(* IEC 61131-3 sources: plc-workspace/projects/FB_MainSequence/03_checks/openplc, 2 files *)

(* ---- FB_MainSequence_OpenPLC.st ---- *)
(* Generated by validation/scripts/sync-semantics.py; edit 02_src/st. *)
FUNCTION FC_MainSequence_BusyPhase : BOOL
VAR_INPUT
    iPhase : INT := 0;
END_VAR

FC_MainSequence_BusyPhase := (iPhase = 1) OR (iPhase = 2) OR (iPhase = 3);

END_FUNCTION

FUNCTION FC_MainSequence_InvalidPhase : BOOL
VAR_INPUT
    iPhase : INT := 0;
END_VAR

FC_MainSequence_InvalidPhase := (iPhase < 0) OR ((iPhase > 3) AND (iPhase <> 900));

END_FUNCTION

FUNCTION FC_MainSequence_StepDone : BOOL
VAR_INPUT
    iPhase : INT := 0;
    xTransportDone : BOOL := FALSE;
    xFlipDone : BOOL := FALSE;
    xOutputDone : BOOL := FALSE;
END_VAR

CASE iPhase OF
    1:
        FC_MainSequence_StepDone := xTransportDone;
    2:
        FC_MainSequence_StepDone := xFlipDone;
    3:
        FC_MainSequence_StepDone := xOutputDone;
    ELSE
        FC_MainSequence_StepDone := FALSE;
END_CASE;

END_FUNCTION

FUNCTION FC_MainSequence_SuccessPhase : INT
VAR_INPUT
    iPhase : INT := 0;
END_VAR

CASE iPhase OF
    1:
        FC_MainSequence_SuccessPhase := 2;
    2:
        FC_MainSequence_SuccessPhase := 3;
    3:
        FC_MainSequence_SuccessPhase := 1;
    ELSE
        FC_MainSequence_SuccessPhase := iPhase;
END_CASE;

END_FUNCTION

FUNCTION FC_MainSequence_TimeoutReached : BOOL
VAR_INPUT
    xBusyPhase : BOOL := FALSE;
    xStepDone : BOOL := FALSE;
    uiStepTimerStat : UINT := 0;
    uiStepTimeoutScans : UINT := 0;
END_VAR

FC_MainSequence_TimeoutReached :=
    xBusyPhase AND
    (NOT xStepDone) AND
    (uiStepTimeoutScans > 0) AND
    ((uiStepTimerStat + 1) >= uiStepTimeoutScans);

END_FUNCTION

FUNCTION FC_MainSequence_NextPhase : INT
VAR_INPUT
    xClearReq : BOOL := FALSE;
    xAbortReq : BOOL := FALSE;
    xFaultLatched : BOOL := FALSE;
    iPhaseStat : INT := 0;
    xInvalidPhase : BOOL := FALSE;
    xStepDone : BOOL := FALSE;
    xTimeoutReached : BOOL := FALSE;
    iSuccessPhase : INT := 0;
    xStartReady : BOOL := FALSE;
END_VAR

IF xClearReq THEN
    FC_MainSequence_NextPhase := 0;
ELSIF xFaultLatched OR xInvalidPhase THEN
    FC_MainSequence_NextPhase := 900;
ELSIF xAbortReq THEN
    FC_MainSequence_NextPhase := 0;
ELSIF iPhaseStat = 0 THEN
    IF xStartReady THEN
        FC_MainSequence_NextPhase := 1;
    ELSE
        FC_MainSequence_NextPhase := 0;
    END_IF;
ELSIF iPhaseStat = 900 THEN
    FC_MainSequence_NextPhase := 900;
ELSIF xInvalidPhase THEN
    FC_MainSequence_NextPhase := 900;
ELSIF xStepDone THEN
    FC_MainSequence_NextPhase := iSuccessPhase;
ELSIF xTimeoutReached THEN
    FC_MainSequence_NextPhase := 900;
ELSE
    FC_MainSequence_NextPhase := iPhaseStat;
END_IF;

END_FUNCTION

FUNCTION FC_MainSequence_NextTimer : UINT
VAR_INPUT
    xResetReq : BOOL := FALSE;
    iPhaseStat : INT := 0;
    xInvalidPhase : BOOL := FALSE;
    xStepDone : BOOL := FALSE;
    xTimeoutReached : BOOL := FALSE;
    xBusyPhase : BOOL := FALSE;
    uiStepTimerStat : UINT := 0;
    uiStepTimeoutScans : UINT := 0;
END_VAR

IF xResetReq OR (iPhaseStat = 0) OR (iPhaseStat = 900) OR xInvalidPhase OR xStepDone OR xTimeoutReached THEN
    FC_MainSequence_NextTimer := 0;
ELSIF xBusyPhase AND (uiStepTimeoutScans > 0) THEN
    FC_MainSequence_NextTimer := uiStepTimerStat + 1;
ELSE
    FC_MainSequence_NextTimer := 0;
END_IF;

END_FUNCTION

FUNCTION FC_MainSequence_NextTimeoutFault : BOOL
VAR_INPUT
    xClearReq : BOOL := FALSE;
    xAbortReq : BOOL := FALSE;
    xTimeoutReached : BOOL := FALSE;
    xTimeoutFaultStat : BOOL := FALSE;
END_VAR

IF xClearReq THEN
    FC_MainSequence_NextTimeoutFault := FALSE;
ELSIF xAbortReq THEN
    FC_MainSequence_NextTimeoutFault := xTimeoutFaultStat;
ELSE
    FC_MainSequence_NextTimeoutFault := xTimeoutFaultStat OR xTimeoutReached;
END_IF;

END_FUNCTION

FUNCTION_BLOCK FB_MainSequence
VAR_INPUT
    xEnable : BOOL := FALSE;
    xEvtStart : BOOL := FALSE;
    xEStop : BOOL := FALSE;
    xStop : BOOL := FALSE;
    xReset : BOOL := FALSE;
    xInitDone : BOOL := FALSE;
    xTransportDone : BOOL := FALSE;
    xFlipDone : BOOL := FALSE;
    xOutputDone : BOOL := FALSE;
    uiStepTimeoutScans : UINT := 8;
END_VAR

VAR_OUTPUT
    iPhase : INT := 0;
    xBeltForward : BOOL := FALSE;
    xBeltReverse : BOOL := FALSE;
    xStartLamp : BOOL := FALSE;
    xResetLamp : BOOL := FALSE;
    xQ1 : BOOL := FALSE;
    xQ2 : BOOL := FALSE;
    xDone : BOOL := FALSE;
    xError : BOOL := FALSE;
    xTimeoutFault : BOOL := FALSE;
    xValid : BOOL := FALSE;
    xBusy : BOOL := FALSE;
    xCommandBusy : BOOL := FALSE;
    xCommandAborted : BOOL := FALSE;
    xTimeoutDiagnostic : BOOL := FALSE;
END_VAR

VAR
    iPhaseStat : INT := 0;
    uiStepTimerStat : UINT := 0;
    xTimeoutFaultStat : BOOL := FALSE;
    xTimeoutDiagnosticStat : BOOL := FALSE;
    xAbortedStat : BOOL := FALSE;
    xEnablePrev : BOOL := FALSE;
    xStartPrev : BOOL := FALSE;
    xResetPrev : BOOL := FALSE;
END_VAR

VAR_TEMP
    iPhasePrev : INT;
    uiStepTimerPrev : UINT;
    xTimeoutFaultPrev : BOOL;
    xDiagnosticPrev : BOOL;
    xAbortedPrev : BOOL;
    xEnableRise : BOOL;
    xStartRise : BOOL;
    xResetRise : BOOL;
    xStopReq : BOOL;
    xResetAccepted : BOOL;
    xClearReq : BOOL;
    xAbortReq : BOOL;
    xInvalidPhase : BOOL;
    xBusyPhase : BOOL;
    xFaultLatched : BOOL;
    xStepDone : BOOL;
    xTimeoutReached : BOOL;
    iPhaseNext : INT;
    uiStepTimerNext : UINT;
    xTimeoutFaultNext : BOOL;
    xDiagnosticNext : BOOL;
    xAbortedNext : BOOL;
    xStartAccepted : BOOL;
    xErrorCore : BOOL;
    xExecAllowed : BOOL;
END_VAR

(* Snapshot persistent internals only; outputs are never used as state. *)
iPhasePrev := iPhaseStat;
uiStepTimerPrev := uiStepTimerStat;
xTimeoutFaultPrev := xTimeoutFaultStat;
xDiagnosticPrev := xTimeoutDiagnosticStat;
xAbortedPrev := xAbortedStat;
xEnableRise := xEnable AND NOT xEnablePrev;
xStartRise := xEvtStart AND NOT xStartPrev;
xResetRise := xReset AND NOT xResetPrev;

(* xEStop is external safety-inhibit feedback, not an F safety function.
   Reset reinitializes a healthy command. Block errors need enable=FALSE. *)
xStopReq := xEStop OR xStop;
xInvalidPhase := FC_MainSequence_InvalidPhase(iPhase := iPhasePrev);
xBusyPhase := FC_MainSequence_BusyPhase(iPhase := iPhasePrev);
xFaultLatched := (iPhasePrev = 900) OR xTimeoutFaultPrev;
xResetAccepted := xEnable AND xResetRise AND NOT xStopReq AND NOT xFaultLatched AND NOT xInvalidPhase;
xClearReq := (NOT xEnable) OR xResetAccepted;
xAbortReq := xStopReq OR xReset;
xStepDone := FC_MainSequence_StepDone(
    iPhase := iPhasePrev,
    xTransportDone := xTransportDone,
    xFlipDone := xFlipDone,
    xOutputDone := xOutputDone
);
xTimeoutReached := FC_MainSequence_TimeoutReached(
    xBusyPhase := xBusyPhase,
    xStepDone := xStepDone,
    uiStepTimerStat := uiStepTimerPrev,
    uiStepTimeoutScans := uiStepTimeoutScans
);

iPhaseNext := FC_MainSequence_NextPhase(
    xClearReq := xClearReq,
    xAbortReq := xAbortReq,
    xFaultLatched := xFaultLatched,
    iPhaseStat := iPhasePrev,
    xInvalidPhase := xInvalidPhase,
    xStepDone := xStepDone,
    xTimeoutReached := xTimeoutReached,
    iSuccessPhase := FC_MainSequence_SuccessPhase(iPhase := iPhasePrev),
    xStartReady := xEnable AND xInitDone AND xStartRise
);
uiStepTimerNext := FC_MainSequence_NextTimer(
    xResetReq := xClearReq OR xAbortReq,
    iPhaseStat := iPhasePrev,
    xInvalidPhase := xInvalidPhase,
    xStepDone := xStepDone,
    xTimeoutReached := xTimeoutReached,
    xBusyPhase := xBusyPhase,
    uiStepTimerStat := uiStepTimerPrev,
    uiStepTimeoutScans := uiStepTimeoutScans
);
xTimeoutFaultNext := FC_MainSequence_NextTimeoutFault(
    xClearReq := xClearReq,
    xAbortReq := xAbortReq,
    xTimeoutReached := xTimeoutReached,
    xTimeoutFaultStat := xTimeoutFaultPrev
);
xStartAccepted := (iPhasePrev = 0) AND (iPhaseNext = 1);

(* Current errors and diagnostic history have separate lifetimes. *)
IF xEnableRise THEN
    xDiagnosticNext := xTimeoutFaultNext;
ELSE
    xDiagnosticNext := xDiagnosticPrev OR xTimeoutFaultNext;
END_IF;
IF xBusyPhase AND (xClearReq OR xAbortReq) THEN
    xAbortedNext := TRUE;
ELSIF (NOT xEnable) OR xResetAccepted OR xStartAccepted THEN
    xAbortedNext := FALSE;
ELSE
    xAbortedNext := xAbortedPrev;
END_IF;
xErrorCore := FC_MainSequence_InvalidPhase(iPhase := iPhaseNext) OR (iPhaseNext = 900);
xExecAllowed := xEnable AND NOT xAbortReq AND NOT xErrorCore;

(* Commit once. Consume input edges on every call, even while inhibited. *)
iPhaseStat := iPhaseNext;
uiStepTimerStat := uiStepTimerNext;
xTimeoutFaultStat := xTimeoutFaultNext;
xTimeoutDiagnosticStat := xDiagnosticNext;
xAbortedStat := xAbortedNext;
xEnablePrev := xEnable;
xStartPrev := xEvtStart;
xResetPrev := xReset;

(* DA008: each output is assigned once and no output is read. *)
iPhase := iPhaseNext;
xError := xErrorCore;
xTimeoutFault := xTimeoutFaultNext;
xBeltForward := xExecAllowed AND ((iPhaseNext = 1) OR (iPhaseNext = 3));
xBeltReverse := FALSE;
xStartLamp := xExecAllowed AND ((iPhaseNext = 2) OR (iPhaseNext = 3));
xResetLamp := xExecAllowed AND (iPhaseNext = 0);
xQ1 := xExecAllowed AND (iPhaseNext = 2);
xQ2 := xExecAllowed AND (iPhaseNext = 3);
xDone := xExecAllowed AND (iPhasePrev = 3) AND xOutputDone AND (iPhaseNext = 1);
xValid := xEnable AND NOT xErrorCore;
xBusy := xEnable AND NOT xErrorCore;
xCommandBusy := xExecAllowed AND FC_MainSequence_BusyPhase(iPhase := iPhaseNext);
xCommandAborted := xAbortedNext;
xTimeoutDiagnostic := xDiagnosticNext;

END_FUNCTION_BLOCK

(* OpenPLC-only test driver. Core definitions are generated from 02_src/st. *)
PROGRAM PLC_PRG
VAR
    fbMain : FB_MainSequence;
    xEnableSim : BOOL := TRUE;
    xEvtStartSim : BOOL := FALSE;
    xEStopSim : BOOL := FALSE;
    xResetSim : BOOL := FALSE;
    xInitDoneSim : BOOL := TRUE;
    xTransportDoneSim : BOOL := FALSE;
    xFlipDoneSim : BOOL := FALSE;
    xOutputDoneSim : BOOL := FALSE;
    uiStepTimeoutScansSim : UINT := 8;

    iObservedPhase : INT := 0;
    xObservedDone : BOOL := FALSE;
    xObservedError : BOOL := FALSE;
    xObservedTimeoutFault : BOOL := FALSE;

    iLastObservedPhase : INT := -1;
    iPhaseDwell : INT := 0;
    iCycleCountInternal : INT := 0;
    iResetCountInternal : INT := 0;
    iScanCountInternal : INT := 0;
    iScenarioCaseInternal : INT := 0;
    iNextScenarioAfterReset : INT := -1;
    iErrorPhaseLatched : INT := 0;

    xDoneLast : BOOL := FALSE;
    xResetPending : BOOL := FALSE;
    xStartPulsePending : BOOL := FALSE;
    xFaultScenarioStarted : BOOL := FALSE;
    xFaultPulseIssued : BOOL := FALSE;
    xRepeatScenarioStarted : BOOL := FALSE;
    iRepeatPulseCount : INT := 0;
    iRepeatBaselineCycle : INT := -1;
    xTimeoutScenarioStarted : BOOL := FALSE;
    xDisablePending : BOOL := FALSE;
END_VAR

VAR
    iPhaseMon AT %MW0 : INT;
    iCycleCountMon AT %MW1 : INT;
    iResetCountMon AT %MW2 : INT;
    iScanCountMon AT %MW3 : INT;
    iScenarioCaseMon AT %MW4 : INT;
    iErrorPhaseMon AT %MW5 : INT;

    xSawPhase0Mon AT %QX0.0 : BOOL;
    xSawPhase1Mon AT %QX0.1 : BOOL;
    xSawPhase2Mon AT %QX0.2 : BOOL;
    xSawPhase3Mon AT %QX0.3 : BOOL;
    xSawDoneMon AT %QX0.4 : BOOL;
    xSawResetReturnMon AT %QX0.5 : BOOL;
    xBehaviorPassMon AT %QX0.6 : BOOL;
    xBehaviorFailMon AT %QX0.7 : BOOL;

    xFaultInterruptPassMon AT %QX1.0 : BOOL;
    xRepeatStartBlockedPassMon AT %QX1.1 : BOOL;
    xTimeoutFailPassMon AT %QX1.2 : BOOL;
    xStartEventRequiredPassMon AT %QX1.3 : BOOL;
    xTimeoutErrorPassMon AT %QX1.4 : BOOL;
END_VAR

iScanCountInternal := iScanCountInternal + 1;
xEvtStartSim := FALSE;
xEStopSim := FALSE;
xResetSim := FALSE;
xTransportDoneSim := FALSE;
xFlipDoneSim := FALSE;
xOutputDoneSim := FALSE;
xEnableSim := TRUE;
xInitDoneSim := TRUE;

IF xDisablePending THEN
    xEnableSim := FALSE;
    xDisablePending := FALSE;
END_IF;

IF xResetPending THEN
    xResetSim := TRUE;
    xResetPending := FALSE;
    iResetCountInternal := iResetCountInternal + 1;
END_IF;

IF xStartPulsePending THEN
    xEvtStartSim := TRUE;
    xStartPulsePending := FALSE;
END_IF;

IF iScenarioCaseInternal = 99 THEN
    xEnableSim := FALSE;
    xInitDoneSim := FALSE;
END_IF;

CASE iScenarioCaseInternal OF
    0:
        IF (iObservedPhase <> 0) AND (NOT xStartEventRequiredPassMon) AND (iCycleCountInternal = 0) THEN
            xBehaviorFailMon := TRUE;
        END_IF;
        IF (iObservedPhase = 0) AND (iPhaseDwell >= 2) AND (NOT xStartEventRequiredPassMon) THEN
            xStartEventRequiredPassMon := TRUE;
            xStartPulsePending := TRUE;
            iScenarioCaseInternal := 1;
        END_IF;

    1:
        CASE iLastObservedPhase OF
            1:
                IF iPhaseDwell >= 2 THEN
                    xTransportDoneSim := TRUE;
                END_IF;
            2:
                IF iPhaseDwell >= 2 THEN
                    xFlipDoneSim := TRUE;
                END_IF;
            3:
                IF iPhaseDwell >= 2 THEN
                    xOutputDoneSim := TRUE;
                END_IF;
        END_CASE;

    2:
        IF (NOT xFaultScenarioStarted) AND (iObservedPhase = 0) AND (iPhaseDwell >= 1) THEN
            xStartPulsePending := TRUE;
            xFaultScenarioStarted := TRUE;
        END_IF;
        IF xFaultScenarioStarted AND (iObservedPhase = 1) AND (iPhaseDwell >= 2) AND (NOT xFaultPulseIssued) THEN
            xEStopSim := TRUE;
            xFaultPulseIssued := TRUE;
        END_IF;

    3:
        IF (NOT xRepeatScenarioStarted) AND (iObservedPhase = 0) AND (iPhaseDwell >= 1) THEN
            xStartPulsePending := TRUE;
            xRepeatScenarioStarted := TRUE;
        END_IF;

        CASE iLastObservedPhase OF
            1:
                IF iPhaseDwell >= 2 THEN
                    xTransportDoneSim := TRUE;
                END_IF;
            2:
                IF iRepeatBaselineCycle < 0 THEN
                    iRepeatBaselineCycle := iCycleCountInternal;
                END_IF;
                IF (iRepeatPulseCount < 3) AND (iPhaseDwell >= (iRepeatPulseCount + 1)) THEN
                    xEvtStartSim := TRUE;
                    iRepeatPulseCount := iRepeatPulseCount + 1;
                END_IF;
                IF (iRepeatPulseCount >= 3) AND (iCycleCountInternal = iRepeatBaselineCycle) THEN
                    xRepeatStartBlockedPassMon := TRUE;
                END_IF;
                IF (iRepeatPulseCount >= 3) AND (iPhaseDwell >= 6) THEN
                    xFlipDoneSim := TRUE;
                END_IF;
            3:
                IF iPhaseDwell >= 2 THEN
                    xOutputDoneSim := TRUE;
                END_IF;
        END_CASE;

    4:
        IF (NOT xTimeoutScenarioStarted) AND (iObservedPhase = 0) AND (iPhaseDwell >= 1) THEN
            xStartPulsePending := TRUE;
            xTimeoutScenarioStarted := TRUE;
        END_IF;
END_CASE;

fbMain(
    xEnable := xEnableSim,
    xEvtStart := xEvtStartSim,
    xEStop := xEStopSim,
    xStop := FALSE,
    xReset := xResetSim,
    xInitDone := xInitDoneSim,
    xTransportDone := xTransportDoneSim,
    xFlipDone := xFlipDoneSim,
    xOutputDone := xOutputDoneSim,
    uiStepTimeoutScans := uiStepTimeoutScansSim
);

iObservedPhase := fbMain.iPhase;
xObservedDone := fbMain.xDone;
xObservedError := fbMain.xError;
xObservedTimeoutFault := fbMain.xTimeoutFault;

IF iObservedPhase = iLastObservedPhase THEN
    iPhaseDwell := iPhaseDwell + 1;
ELSE
    iPhaseDwell := 0;
    iLastObservedPhase := iObservedPhase;
END_IF;

CASE iObservedPhase OF
    0:
        xSawPhase0Mon := TRUE;
    1:
        xSawPhase1Mon := TRUE;
    2:
        xSawPhase2Mon := TRUE;
    3:
        xSawPhase3Mon := TRUE;
END_CASE;

IF (iScenarioCaseInternal = 2) AND xFaultPulseIssued AND (iObservedPhase = 0) AND
   (NOT fbMain.xBeltForward) AND (NOT fbMain.xStartLamp) AND
   (NOT fbMain.xQ1) AND (NOT fbMain.xQ2) THEN
    xFaultInterruptPassMon := TRUE;
    iScenarioCaseInternal := 3;
    xFaultScenarioStarted := FALSE;
    xFaultPulseIssued := FALSE;
END_IF;

IF (iScenarioCaseInternal = 3) AND (iRepeatPulseCount > 0) AND (iRepeatPulseCount < 3) AND
   (iObservedPhase <> 2) THEN
    xBehaviorFailMon := TRUE;
END_IF;

IF xObservedDone AND (NOT xDoneLast) THEN
    xSawDoneMon := TRUE;
    iCycleCountInternal := iCycleCountInternal + 1;
    CASE iScenarioCaseInternal OF
        1:
            iNextScenarioAfterReset := 2;
            xResetPending := TRUE;
        3:
            iNextScenarioAfterReset := 4;
            xResetPending := TRUE;
    END_CASE;
END_IF;
xDoneLast := xObservedDone;

IF (iScenarioCaseInternal = 4) AND (iObservedPhase = 900) AND xObservedError AND xObservedTimeoutFault THEN
    xTimeoutErrorPassMon := TRUE;
    xTimeoutFailPassMon := TRUE;
    iErrorPhaseLatched := 900;
    iNextScenarioAfterReset := 99;
    xDisablePending := TRUE;
END_IF;

IF (iNextScenarioAfterReset >= 0) AND (iObservedPhase = 0) THEN
    xSawResetReturnMon := TRUE;
    iScenarioCaseInternal := iNextScenarioAfterReset;
    iNextScenarioAfterReset := -1;
    iRepeatPulseCount := 0;
    iRepeatBaselineCycle := -1;
END_IF;

IF xObservedError AND NOT ((iObservedPhase = 900) AND xObservedTimeoutFault) THEN
    xBehaviorFailMon := TRUE;
END_IF;

IF (NOT xBehaviorPassMon) AND
   xSawPhase0Mon AND xSawPhase1Mon AND xSawPhase2Mon AND xSawPhase3Mon AND
   xSawDoneMon AND xSawResetReturnMon AND
   xFaultInterruptPassMon AND xRepeatStartBlockedPassMon AND xTimeoutFailPassMon AND
   xStartEventRequiredPassMon AND xTimeoutErrorPassMon AND
   (iObservedPhase = 0) AND (iScenarioCaseInternal = 99) THEN
    xBehaviorPassMon := TRUE;
    xBehaviorFailMon := FALSE;
END_IF;

IF (NOT xBehaviorPassMon) AND (iScanCountInternal > 800) THEN
    xBehaviorFailMon := TRUE;
END_IF;

iPhaseMon := iObservedPhase;
iCycleCountMon := iCycleCountInternal;
iResetCountMon := iResetCountInternal;
iScanCountMon := iScanCountInternal;
iScenarioCaseMon := iScenarioCaseInternal;
iErrorPhaseMon := iErrorPhaseLatched;

END_PROGRAM

CONFIGURATION Config0

  RESOURCE Res0 ON PLC
    TASK Main(INTERVAL := T#50ms, PRIORITY := 0);
    PROGRAM Inst0 WITH Main : PLC_PRG;
  END_RESOURCE
END_CONFIGURATION

(* ---- driver.st ---- *)
(* OpenPLC-only test driver. Core definitions are generated from 02_src/st. *)
PROGRAM PLC_PRG
VAR
    fbMain : FB_MainSequence;
    xEnableSim : BOOL := TRUE;
    xEvtStartSim : BOOL := FALSE;
    xEStopSim : BOOL := FALSE;
    xResetSim : BOOL := FALSE;
    xInitDoneSim : BOOL := TRUE;
    xTransportDoneSim : BOOL := FALSE;
    xFlipDoneSim : BOOL := FALSE;
    xOutputDoneSim : BOOL := FALSE;
    uiStepTimeoutScansSim : UINT := 8;

    iObservedPhase : INT := 0;
    xObservedDone : BOOL := FALSE;
    xObservedError : BOOL := FALSE;
    xObservedTimeoutFault : BOOL := FALSE;

    iLastObservedPhase : INT := -1;
    iPhaseDwell : INT := 0;
    iCycleCountInternal : INT := 0;
    iResetCountInternal : INT := 0;
    iScanCountInternal : INT := 0;
    iScenarioCaseInternal : INT := 0;
    iNextScenarioAfterReset : INT := -1;
    iErrorPhaseLatched : INT := 0;

    xDoneLast : BOOL := FALSE;
    xResetPending : BOOL := FALSE;
    xStartPulsePending : BOOL := FALSE;
    xFaultScenarioStarted : BOOL := FALSE;
    xFaultPulseIssued : BOOL := FALSE;
    xRepeatScenarioStarted : BOOL := FALSE;
    iRepeatPulseCount : INT := 0;
    iRepeatBaselineCycle : INT := -1;
    xTimeoutScenarioStarted : BOOL := FALSE;
    xDisablePending : BOOL := FALSE;
END_VAR

VAR
    iPhaseMon AT %MW0 : INT;
    iCycleCountMon AT %MW1 : INT;
    iResetCountMon AT %MW2 : INT;
    iScanCountMon AT %MW3 : INT;
    iScenarioCaseMon AT %MW4 : INT;
    iErrorPhaseMon AT %MW5 : INT;

    xSawPhase0Mon AT %QX0.0 : BOOL;
    xSawPhase1Mon AT %QX0.1 : BOOL;
    xSawPhase2Mon AT %QX0.2 : BOOL;
    xSawPhase3Mon AT %QX0.3 : BOOL;
    xSawDoneMon AT %QX0.4 : BOOL;
    xSawResetReturnMon AT %QX0.5 : BOOL;
    xBehaviorPassMon AT %QX0.6 : BOOL;
    xBehaviorFailMon AT %QX0.7 : BOOL;

    xFaultInterruptPassMon AT %QX1.0 : BOOL;
    xRepeatStartBlockedPassMon AT %QX1.1 : BOOL;
    xTimeoutFailPassMon AT %QX1.2 : BOOL;
    xStartEventRequiredPassMon AT %QX1.3 : BOOL;
    xTimeoutErrorPassMon AT %QX1.4 : BOOL;
END_VAR

iScanCountInternal := iScanCountInternal + 1;
xEvtStartSim := FALSE;
xEStopSim := FALSE;
xResetSim := FALSE;
xTransportDoneSim := FALSE;
xFlipDoneSim := FALSE;
xOutputDoneSim := FALSE;
xEnableSim := TRUE;
xInitDoneSim := TRUE;

IF xDisablePending THEN
    xEnableSim := FALSE;
    xDisablePending := FALSE;
END_IF;

IF xResetPending THEN
    xResetSim := TRUE;
    xResetPending := FALSE;
    iResetCountInternal := iResetCountInternal + 1;
END_IF;

IF xStartPulsePending THEN
    xEvtStartSim := TRUE;
    xStartPulsePending := FALSE;
END_IF;

IF iScenarioCaseInternal = 99 THEN
    xEnableSim := FALSE;
    xInitDoneSim := FALSE;
END_IF;

CASE iScenarioCaseInternal OF
    0:
        IF (iObservedPhase <> 0) AND (NOT xStartEventRequiredPassMon) AND (iCycleCountInternal = 0) THEN
            xBehaviorFailMon := TRUE;
        END_IF;
        IF (iObservedPhase = 0) AND (iPhaseDwell >= 2) AND (NOT xStartEventRequiredPassMon) THEN
            xStartEventRequiredPassMon := TRUE;
            xStartPulsePending := TRUE;
            iScenarioCaseInternal := 1;
        END_IF;

    1:
        CASE iLastObservedPhase OF
            1:
                IF iPhaseDwell >= 2 THEN
                    xTransportDoneSim := TRUE;
                END_IF;
            2:
                IF iPhaseDwell >= 2 THEN
                    xFlipDoneSim := TRUE;
                END_IF;
            3:
                IF iPhaseDwell >= 2 THEN
                    xOutputDoneSim := TRUE;
                END_IF;
        END_CASE;

    2:
        IF (NOT xFaultScenarioStarted) AND (iObservedPhase = 0) AND (iPhaseDwell >= 1) THEN
            xStartPulsePending := TRUE;
            xFaultScenarioStarted := TRUE;
        END_IF;
        IF xFaultScenarioStarted AND (iObservedPhase = 1) AND (iPhaseDwell >= 2) AND (NOT xFaultPulseIssued) THEN
            xEStopSim := TRUE;
            xFaultPulseIssued := TRUE;
        END_IF;

    3:
        IF (NOT xRepeatScenarioStarted) AND (iObservedPhase = 0) AND (iPhaseDwell >= 1) THEN
            xStartPulsePending := TRUE;
            xRepeatScenarioStarted := TRUE;
        END_IF;

        CASE iLastObservedPhase OF
            1:
                IF iPhaseDwell >= 2 THEN
                    xTransportDoneSim := TRUE;
                END_IF;
            2:
                IF iRepeatBaselineCycle < 0 THEN
                    iRepeatBaselineCycle := iCycleCountInternal;
                END_IF;
                IF (iRepeatPulseCount < 3) AND (iPhaseDwell >= (iRepeatPulseCount + 1)) THEN
                    xEvtStartSim := TRUE;
                    iRepeatPulseCount := iRepeatPulseCount + 1;
                END_IF;
                IF (iRepeatPulseCount >= 3) AND (iCycleCountInternal = iRepeatBaselineCycle) THEN
                    xRepeatStartBlockedPassMon := TRUE;
                END_IF;
                IF (iRepeatPulseCount >= 3) AND (iPhaseDwell >= 6) THEN
                    xFlipDoneSim := TRUE;
                END_IF;
            3:
                IF iPhaseDwell >= 2 THEN
                    xOutputDoneSim := TRUE;
                END_IF;
        END_CASE;

    4:
        IF (NOT xTimeoutScenarioStarted) AND (iObservedPhase = 0) AND (iPhaseDwell >= 1) THEN
            xStartPulsePending := TRUE;
            xTimeoutScenarioStarted := TRUE;
        END_IF;
END_CASE;

fbMain(
    xEnable := xEnableSim,
    xEvtStart := xEvtStartSim,
    xEStop := xEStopSim,
    xStop := FALSE,
    xReset := xResetSim,
    xInitDone := xInitDoneSim,
    xTransportDone := xTransportDoneSim,
    xFlipDone := xFlipDoneSim,
    xOutputDone := xOutputDoneSim,
    uiStepTimeoutScans := uiStepTimeoutScansSim
);

iObservedPhase := fbMain.iPhase;
xObservedDone := fbMain.xDone;
xObservedError := fbMain.xError;
xObservedTimeoutFault := fbMain.xTimeoutFault;

IF iObservedPhase = iLastObservedPhase THEN
    iPhaseDwell := iPhaseDwell + 1;
ELSE
    iPhaseDwell := 0;
    iLastObservedPhase := iObservedPhase;
END_IF;

CASE iObservedPhase OF
    0:
        xSawPhase0Mon := TRUE;
    1:
        xSawPhase1Mon := TRUE;
    2:
        xSawPhase2Mon := TRUE;
    3:
        xSawPhase3Mon := TRUE;
END_CASE;

IF (iScenarioCaseInternal = 2) AND xFaultPulseIssued AND (iObservedPhase = 0) AND
   (NOT fbMain.xBeltForward) AND (NOT fbMain.xStartLamp) AND
   (NOT fbMain.xQ1) AND (NOT fbMain.xQ2) THEN
    xFaultInterruptPassMon := TRUE;
    iScenarioCaseInternal := 3;
    xFaultScenarioStarted := FALSE;
    xFaultPulseIssued := FALSE;
END_IF;

IF (iScenarioCaseInternal = 3) AND (iRepeatPulseCount > 0) AND (iRepeatPulseCount < 3) AND
   (iObservedPhase <> 2) THEN
    xBehaviorFailMon := TRUE;
END_IF;

IF xObservedDone AND (NOT xDoneLast) THEN
    xSawDoneMon := TRUE;
    iCycleCountInternal := iCycleCountInternal + 1;
    CASE iScenarioCaseInternal OF
        1:
            iNextScenarioAfterReset := 2;
            xResetPending := TRUE;
        3:
            iNextScenarioAfterReset := 4;
            xResetPending := TRUE;
    END_CASE;
END_IF;
xDoneLast := xObservedDone;

IF (iScenarioCaseInternal = 4) AND (iObservedPhase = 900) AND xObservedError AND xObservedTimeoutFault THEN
    xTimeoutErrorPassMon := TRUE;
    xTimeoutFailPassMon := TRUE;
    iErrorPhaseLatched := 900;
    iNextScenarioAfterReset := 99;
    xDisablePending := TRUE;
END_IF;

IF (iNextScenarioAfterReset >= 0) AND (iObservedPhase = 0) THEN
    xSawResetReturnMon := TRUE;
    iScenarioCaseInternal := iNextScenarioAfterReset;
    iNextScenarioAfterReset := -1;
    iRepeatPulseCount := 0;
    iRepeatBaselineCycle := -1;
END_IF;

IF xObservedError AND NOT ((iObservedPhase = 900) AND xObservedTimeoutFault) THEN
    xBehaviorFailMon := TRUE;
END_IF;

IF (NOT xBehaviorPassMon) AND
   xSawPhase0Mon AND xSawPhase1Mon AND xSawPhase2Mon AND xSawPhase3Mon AND
   xSawDoneMon AND xSawResetReturnMon AND
   xFaultInterruptPassMon AND xRepeatStartBlockedPassMon AND xTimeoutFailPassMon AND
   xStartEventRequiredPassMon AND xTimeoutErrorPassMon AND
   (iObservedPhase = 0) AND (iScenarioCaseInternal = 99) THEN
    xBehaviorPassMon := TRUE;
    xBehaviorFailMon := FALSE;
END_IF;

IF (NOT xBehaviorPassMon) AND (iScanCountInternal > 800) THEN
    xBehaviorFailMon := TRUE;
END_IF;

iPhaseMon := iObservedPhase;
iCycleCountMon := iCycleCountInternal;
iResetCountMon := iResetCountInternal;
iScanCountMon := iScanCountInternal;
iScenarioCaseMon := iScenarioCaseInternal;
iErrorPhaseMon := iErrorPhaseLatched;

END_PROGRAM

CONFIGURATION Config0

  RESOURCE Res0 ON PLC
    TASK Main(INTERVAL := T#50ms, PRIORITY := 0);
    PROGRAM Inst0 WITH Main : PLC_PRG;
  END_RESOURCE
END_CONFIGURATION
